// TIA Portal V16 export
// export: Created 2023-06-21T17:06:28.6166611Z, ExportSetting WithDefaults, DisplayName Totally Integrated Automation Portal, DisplayVersion V16 Update 4, DisplayName TIA Portal Version Control Interface, DisplayVersion V16 Update 2, DisplayName TIA Portal Openness, DisplayVersion V16 Update 4, DisplayName SINAMICS Startdrive Advanced, DisplayVersion V16, DisplayName SINAMICS Startdrive G130, G150, S120, S150, SINAMICS MV, S210, DisplayVersion V16, DisplayName SINAMICS Startdrive G110M, G120, G120C, G120D, G120P, DisplayVersion V16, DisplayName STEP 7 Professional, DisplayVersion V16 Update 4, DisplayName STEP 7 Safety, DisplayVersion V16, DisplayName Soft Starter ES, DisplayVersion V16, DisplayName WinCC Advanced, DisplayVersion V16 Update 4
DATA_BLOCK "Modbus_Send_Receive"   // DB10
{ S7_Optimized_Access := 'FALSE' }
VERSION : 0.1
// stored: AutoNumber true, DBAccessibleFromOPCUA true, IsOnlyStoredInLoadMemory false, IsWriteProtectedInAS false
   VAR
      "30001" : Word;
      "30002" : Word;   // COMM_OK = 3FFF
      "32001" : Word;   // STS_UNIT_01
      "32002" : Word;   // OPER_UNIT_01
      "32003" : Word;   // SP_UNIT_01
      "32004" : Word;   // ERROR_UNIT_01
      "32005" : Word;   // PV_UNIT_01
      "32006" : Word;   // SERROR_UNIT_01
      "32007" : Word;   // STS_UNIT_02
      "32008" : Word;   // OPER_UNIT_02
      "32009" : Word;   // SP_UNIT_02
      "32010" : Word;   // ERROR_UNIT_02
      "32011" : Word;   // PV_UNIT_02
      "32012" : Word;   // SERROR_UNIT_02
      "32013" : Word;
      "32014" : Word;
      "32015" : Word;
      "32016" : Word;
      "32017" : Word;
      "32018" : Word;
      "32019" : Word;
      "32020" : Word;
      "32021" : Word;
      "32022" : Word;
      "32023" : Word;
      "32024" : Word;
      "32025" : Word;
      "32026" : Word;
      "32027" : Word;
      "32028" : Word;
      "32029" : Word;
      "32030" : Word;
      "32031" : Word;
      "32032" : Word;
      "32033" : Word;
      "32034" : Word;
      "32035" : Word;
      "32036" : Word;
      "32037" : Word;
      "32038" : Word;
      "32039" : Word;
      "32040" : Word;
      "32041" : Word;
      "32042" : Word;
      "32043" : Word;
      "32044" : Word;
      "32045" : Word;
      "32046" : Word;
      "32047" : Word;
      "32048" : Word;
      "32049" : Word;
      "32050" : Word;
      "32051" : Word;
      "32052" : Word;
      "32053" : Word;
      "32054" : Word;
      "32055" : Word;
      "32056" : Word;
      "32057" : Word;
      "32058" : Word;
      "32059" : Word;
      "32060" : Word;
      "32061" : Word;
      "32062" : Word;
      "32063" : Word;
      "32064" : Word;
      "32065" : Word;
      "32066" : Word;
      "32067" : Word;
      "32068" : Word;
      "32069" : Word;
      "32070" : Word;
      "32071" : Word;
      "32072" : Word;
      "32073" : Word;
      "32074" : Word;
      "32075" : Word;
      "32076" : Word;
      "32077" : Word;
      "32078" : Word;
      "32079" : Word;
      "32080" : Word;
      "32081" : Word;
      "32082" : Word;
      "32083" : Word;
      "32084" : Word;
      "40001" : Word;   // COMM
      "42001" : Word;   // STS
      "42002" : Word;   // OPER_MODE
      "42003" : Word;   // SP
      "42004" : Word;   // STS
      "42005" : Word;   // OPER_MODE
      "42006" : Word;   // SP
      "42007" : Word;   // STS
      "42008" : Word;   // OPER_MODE
      "42009" : Word;   // SP
      "42010" : Word;   // STS
      "42011" : Word;   // OPER_MODE
      "42012" : Word;   // SP
      "42013" : Word;   // STS
      "42014" : Word;   // OPER_MODE
      "42015" : Word;   // SP
      "42016" : Word;   // STS
      "42017" : Word;   // OPER_MODE
      "42018" : Word;   // SP
      "42019" : Word;   // STS
      "42020" : Word;   // OPER_MODE
      "42021" : Word;   // SP
      "42022" : Word;   // STS
      "42023" : Word;   // OPER_MODE
      "42024" : Word;   // SP
      "42025" : Word;   // STS
      "42026" : Word;   // OPER_MODE
      "42027" : Word;   // SP
      "42028" : Word;   // STS
      "42029" : Word;   // OPER_MODE
      "42030" : Word;   // SP
      "42031" : Word;   // STS
      "42032" : Word;   // OPER_MODE
      "42033" : Word;   // SP
      "42034" : Word;   // STS
      "42035" : Word;   // OPER_MODE
      "42036" : Word;   // SP
      "42037" : Word;   // STS
      "42038" : Word;   // OPER_MODE
      "42039" : Word;   // SP
      "42040" : Word;   // STS
      "42041" : Word;   // OPER_MODE
      "42042" : Word;   // SP
      Extrusora_1 : Struct
         Ligado : Bool;
         Fan : Bool;
         Heating : Bool;
         Cooling : Bool;
         Sts_Fan : Bool;
         Sts_Heating : Bool;
         Sts_Cooling : Bool;
         Slave : Bool;
         Master : Bool;
         SP : Real;
         PV : Real;
      END_STRUCT;
      Extrusora_2 : Struct
         Ligado : Bool;
         Fan : Bool;
         Heating : Bool;
         Cooling : Bool;
         Sts_Fan : Bool;
         Sts_Heating : Bool;
         Sts_Cooling : Bool;
         Slave : Bool;
         Master : Bool;
         SP : Real;
         PV : Real;
      END_STRUCT;
      Extrusora_3 : Struct
         Ligado : Bool;
         Fan : Bool;
         Heating : Bool;
         Cooling : Bool;
         Sts_Fan : Bool;
         Sts_Heating : Bool;
         Sts_Cooling : Bool;
         Slave : Bool;
         Master : Bool;
         SP : Real;
         PV : Real;
      END_STRUCT;
      Extrusora_4 : Struct
         Ligado : Bool;
         Fan : Bool;
         Heating : Bool;
         Cooling : Bool;
         Sts_Fan : Bool;
         Sts_Heating : Bool;
         Sts_Cooling : Bool;
         Slave : Bool;
         Master : Bool;
         SP : Real;
         PV : Real;
      END_STRUCT;
      Extrusora_5 : Struct
         Ligado : Bool;
         Fan : Bool;
         Heating : Bool;
         Cooling : Bool;
         Sts_Fan : Bool;
         Sts_Heating : Bool;
         Sts_Cooling : Bool;
         Slave : Bool;
         Master : Bool;
         SP : Real;
         PV : Real;
      END_STRUCT;
      Extrusora_6 : Struct
         Ligado : Bool;
         Fan : Bool;
         Heating : Bool;
         Cooling : Bool;
         Sts_Fan : Bool;
         Sts_Heating : Bool;
         Sts_Cooling : Bool;
         Slave : Bool;
         Master : Bool;
         SP : Real;
         PV : Real;
      END_STRUCT;
      Extrusora_7 : Struct
         Ligado : Bool;
         Fan : Bool;
         Heating : Bool;
         Cooling : Bool;
         Sts_Fan : Bool;
         Sts_Heating : Bool;
         Sts_Cooling : Bool;
         Slave : Bool;
         Master : Bool;
         SP : Real;
         PV : Real;
      END_STRUCT;
      Extrusora_8 : Struct
         Ligado : Bool;
         Fan : Bool;
         Heating : Bool;
         Cooling : Bool;
         Sts_Fan : Bool;
         Sts_Heating : Bool;
         Sts_Cooling : Bool;
         Slave : Bool;
         Master : Bool;
         SP : Real;
         PV : Real;
      END_STRUCT;
      Extrusora_9 : Struct
         Ligado : Bool;
         Fan : Bool;
         Heating : Bool;
         Cooling : Bool;
         Sts_Fan : Bool;
         Sts_Heating : Bool;
         Sts_Cooling : Bool;
         Slave : Bool;
         Master : Bool;
         SP : Real;
         PV : Real;
      END_STRUCT;
      Extrusora_10 : Struct
         Ligado : Bool;
         Fan : Bool;
         Heating : Bool;
         Cooling : Bool;
         Sts_Fan : Bool;
         Sts_Heating : Bool;
         Sts_Cooling : Bool;
         Slave : Bool;
         Master : Bool;
         SP : Real;
         PV : Real;
      END_STRUCT;
      Extrusora_11 : Struct
         Ligado : Bool;
         Fan : Bool;
         Heating : Bool;
         Cooling : Bool;
         Sts_Fan : Bool;
         Sts_Heating : Bool;
         Sts_Cooling : Bool;
         Slave : Bool;
         Master : Bool;
         SP : Real;
         PV : Real;
      END_STRUCT;
      Extrusora_12 : Struct
         Ligado : Bool;
         Fan : Bool;
         Heating : Bool;
         Cooling : Bool;
         Sts_Fan : Bool;
         Sts_Heating : Bool;
         Sts_Cooling : Bool;
         Slave : Bool;
         Master : Bool;
         SP : Real;
         PV : Real;
      END_STRUCT;
      Extrusora_13 : Struct
         Ligado : Bool;
         Fan : Bool;
         Heating : Bool;
         Cooling : Bool;
         Sts_Fan : Bool;
         Sts_Heating : Bool;
         Sts_Cooling : Bool;
         Slave : Bool;
         Master : Bool;
         SP : Real;
         PV : Real;
      END_STRUCT;
      Extrusora_14 : Struct
         Ligado : Bool;
         Fan : Bool;
         Heating : Bool;
         Cooling : Bool;
         Sts_Fan : Bool;
         Sts_Heating : Bool;
         Sts_Cooling : Bool;
         Slave : Bool;
         Master : Bool;
         SP : Real;
         PV : Real;
      END_STRUCT;
      Malfunction_1 : Bool;
      Malfunction_2 : Bool;
      Malfunction_3 : Bool;
      Malfunction_4 : Bool;
      Malfunction_5 : Bool;
      Malfunction_6 : Bool;
      Malfunction_7 : Bool;
      Malfunction_8 : Bool;
      Malfunction_9 : Bool;
      Malfunction_10 : Bool;
      Malfunction_11 : Bool;
      Malfunction_12 : Bool;
      Malfunction_13 : Bool;
      Malfunction_14 : Bool;
   END_VAR
BEGIN
END_DATA_BLOCK
